// TIA Portal V18 export
FUNCTION "VerticalBeam_Main" : Void   // FC7, LAD
{ S7_Optimized_Access := 'TRUE' }
VERSION : 0.1
// stored: AutoNumber true, IsIECCheckEnabled false, SetENOAutomatically false, UDAEnableTagReadback false
BEGIN

REGION Network 1: 区域搜索
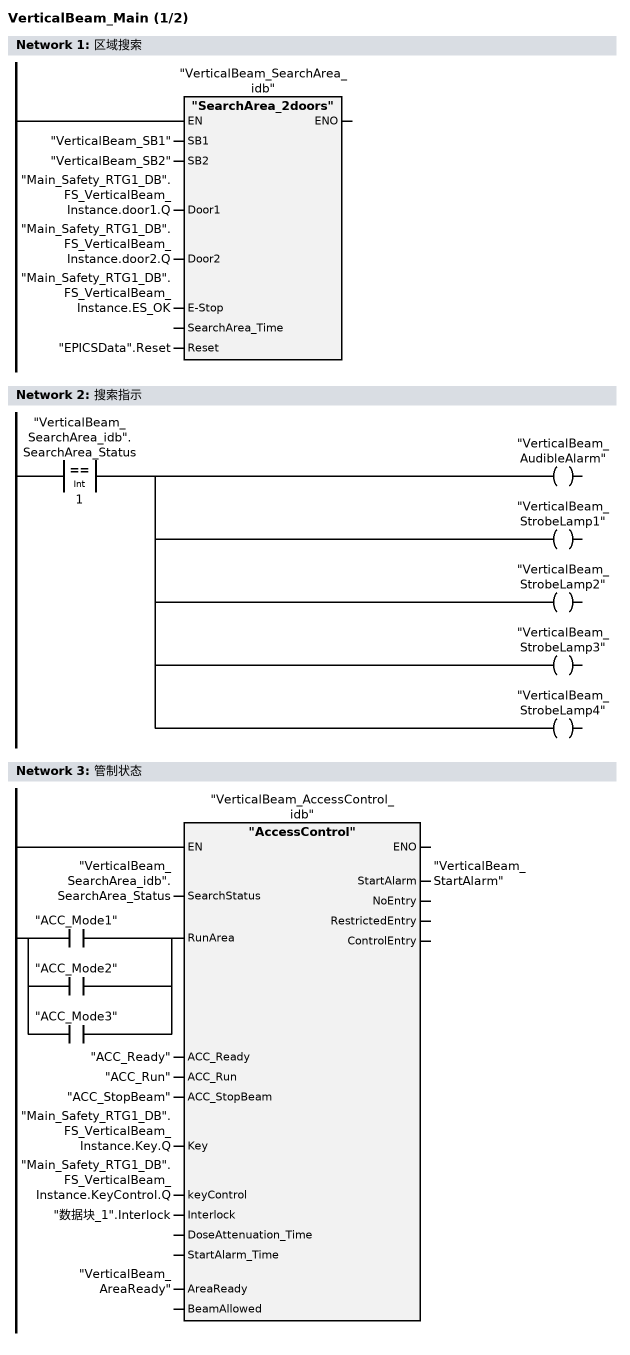
   RUNG wire#powerrail
      "VerticalBeam_SearchArea_idb"(SB1 := "VerticalBeam_SB1", SB2 := "VerticalBeam_SB2", Door1 := "Main_Safety_RTG1_DB".FS_VerticalBeam_Instance.door1.Q, Door2 := "Main_Safety_RTG1_DB".FS_VerticalBeam_Instance.door2.Q, "E-Stop" := "Main_Safety_RTG1_DB".FS_VerticalBeam_Instance.ES_OK, SearchArea_Time :=, Reset := "EPICSData".Reset)
   END_RUNG
   // the same network as SCL:
   "VerticalBeam_SearchArea_idb"(SB1 := "VerticalBeam_SB1",   // "SearchArea_2doors"
                           SB2 := "VerticalBeam_SB2",
                           Door1 := "Main_Safety_RTG1_DB".FS_VerticalBeam_Instance.door1.Q,
                           Door2 := "Main_Safety_RTG1_DB".FS_VerticalBeam_Instance.door2.Q,
                           "E-Stop" := "Main_Safety_RTG1_DB".FS_VerticalBeam_Instance.ES_OK,
                           Reset := "EPICSData".Reset);
END_REGION

REGION Network 2: 搜索指示
   RUNG wire#powerrail
      { S7_Templates := "SrcType := Int" } EQ_Contact(in1 := "VerticalBeam_SearchArea_idb".SearchArea_Status, in2 := 1)
      wire#w1
      Coil( "VerticalBeam_AudibleAlarm" )
   END_RUNG
   RUNG wire#w1
      Coil( "VerticalBeam_StrobeLamp1" )
   END_RUNG
   RUNG wire#w1
      Coil( "VerticalBeam_StrobeLamp2" )
   END_RUNG
   RUNG wire#w1
      Coil( "VerticalBeam_StrobeLamp3" )
   END_RUNG
   RUNG wire#w1
      Coil( "VerticalBeam_StrobeLamp4" )
   END_RUNG
   // the same network as SCL:
   "VerticalBeam_AudibleAlarm" := "VerticalBeam_SearchArea_idb".SearchArea_Status = 1;
   "VerticalBeam_StrobeLamp1" := "VerticalBeam_AudibleAlarm";
   "VerticalBeam_StrobeLamp2" := "VerticalBeam_AudibleAlarm";
   "VerticalBeam_StrobeLamp3" := "VerticalBeam_AudibleAlarm";
   "VerticalBeam_StrobeLamp4" := "VerticalBeam_AudibleAlarm";
END_REGION

REGION Network 3: 管制状态
   RUNG wire#powerrail
      "VerticalBeam_AccessControl_idb"(RunArea := wire#w1, SearchStatus := "VerticalBeam_SearchArea_idb".SearchArea_Status, ACC_Ready := "ACC_Ready", ACC_Run := "ACC_Run", ACC_StopBeam := "ACC_StopBeam", Key := "Main_Safety_RTG1_DB".FS_VerticalBeam_Instance.Key.Q, keyControl := "Main_Safety_RTG1_DB".FS_VerticalBeam_Instance.KeyControl.Q, Interlock := "数据块_1".Interlock, DoseAttenuation_Time :=, StartAlarm_Time :=, AreaReady := "VerticalBeam_AreaReady", BeamAllowed :=, StartAlarm => "VerticalBeam_StartAlarm", NoEntry =>, RestrictedEntry =>, ControlEntry =>)
   END_RUNG
   RUNG wire#powerrail
      Contact( "ACC_Mode1" )
   END_RUNG wire#w1
   RUNG wire#powerrail
      Contact( "ACC_Mode2" )
   END_RUNG wire#w1
   RUNG wire#powerrail
      Contact( "ACC_Mode3" )
   END_RUNG wire#w1
   // the same network as SCL:
   "VerticalBeam_AccessControl_idb"(SearchStatus := "VerticalBeam_SearchArea_idb".SearchArea_Status,   // "AccessControl"
                           RunArea := "ACC_Mode1" OR "ACC_Mode2" OR "ACC_Mode3",
                           ACC_Ready := "ACC_Ready",
                           ACC_Run := "ACC_Run",
                           ACC_StopBeam := "ACC_StopBeam",
                           Key := "Main_Safety_RTG1_DB".FS_VerticalBeam_Instance.Key.Q,
                           keyControl := "Main_Safety_RTG1_DB".FS_VerticalBeam_Instance.KeyControl.Q,
                           Interlock := "数据块_1".Interlock,
                           AreaReady := "VerticalBeam_AreaReady",
                           StartAlarm => "VerticalBeam_StartAlarm");
END_REGION

REGION Network 4: 管制输出
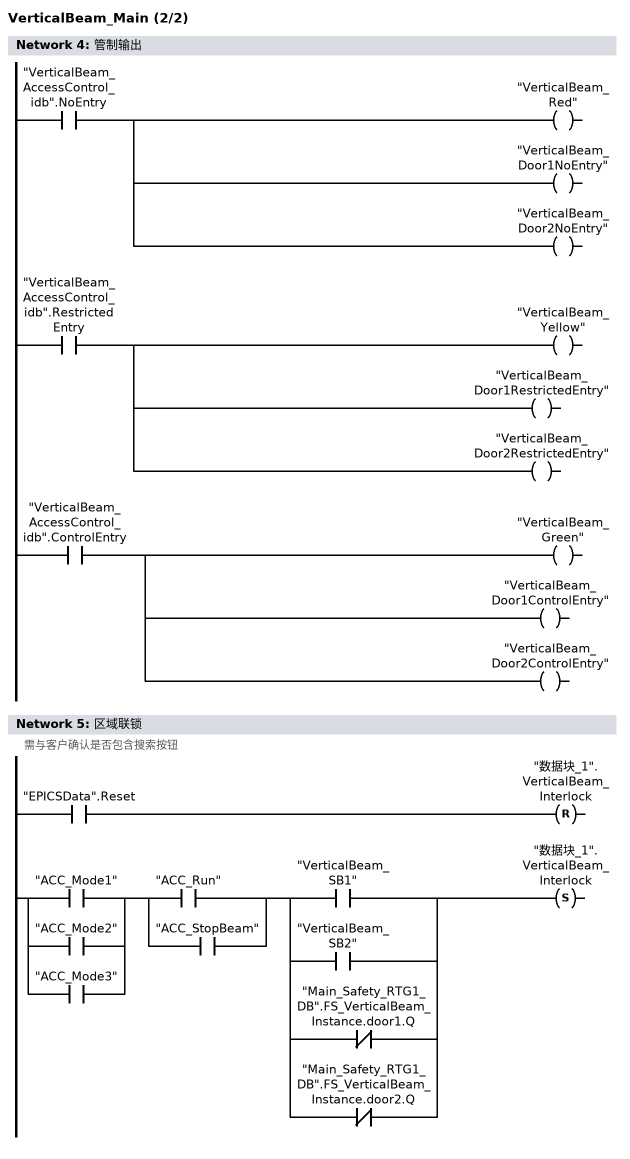
   RUNG wire#powerrail
      Contact( "VerticalBeam_AccessControl_idb".NoEntry )
      wire#w1
      Coil( "VerticalBeam_Red" )
   END_RUNG
   RUNG wire#w1
      Coil( "VerticalBeam_Door1NoEntry" )
   END_RUNG
   RUNG wire#w1
      Coil( "VerticalBeam_Door2NoEntry" )
   END_RUNG
   RUNG wire#powerrail
      Contact( "VerticalBeam_AccessControl_idb".RestrictedEntry )
      wire#w2
      Coil( "VerticalBeam_Yellow" )
   END_RUNG
   RUNG wire#w2
      Coil( "VerticalBeam_Door1RestrictedEntry" )
   END_RUNG
   RUNG wire#w2
      Coil( "VerticalBeam_Door2RestrictedEntry" )
   END_RUNG
   RUNG wire#powerrail
      Contact( "VerticalBeam_AccessControl_idb".ControlEntry )
      wire#w3
      Coil( "VerticalBeam_Green" )
   END_RUNG
   RUNG wire#w3
      Coil( "VerticalBeam_Door1ControlEntry" )
   END_RUNG
   RUNG wire#w3
      Coil( "VerticalBeam_Door2ControlEntry" )
   END_RUNG
   // the same network as SCL:
   "VerticalBeam_Red" := "VerticalBeam_AccessControl_idb".NoEntry;
   "VerticalBeam_Door1NoEntry" := "VerticalBeam_AccessControl_idb".NoEntry;
   "VerticalBeam_Door2NoEntry" := "VerticalBeam_AccessControl_idb".NoEntry;
   "VerticalBeam_Yellow" := "VerticalBeam_AccessControl_idb".RestrictedEntry;
   "VerticalBeam_Door1RestrictedEntry" := "VerticalBeam_AccessControl_idb".RestrictedEntry;
   "VerticalBeam_Door2RestrictedEntry" := "VerticalBeam_AccessControl_idb".RestrictedEntry;
   "VerticalBeam_Green" := "VerticalBeam_AccessControl_idb".ControlEntry;
   "VerticalBeam_Door1ControlEntry" := "VerticalBeam_AccessControl_idb".ControlEntry;
   "VerticalBeam_Door2ControlEntry" := "VerticalBeam_AccessControl_idb".ControlEntry;
END_REGION

REGION Network 5: 区域联锁
   // 需与客户确认是否包含搜索按钮
   RUNG wire#powerrail
      Contact( "EPICSData".Reset )
      R_Coil( "数据块_1".VerticalBeam_Interlock )
   END_RUNG
   RUNG wire#powerrail
      Contact( "ACC_Mode1" )
      wire#w1
      Contact( "ACC_Run" )
      wire#w2
      Contact( "VerticalBeam_SB1" )
      wire#w3
      S_Coil( "数据块_1".VerticalBeam_Interlock )
   END_RUNG
   RUNG wire#powerrail
      Contact( "ACC_Mode2" )
   END_RUNG wire#w1
   RUNG wire#powerrail
      Contact( "ACC_Mode3" )
   END_RUNG wire#w1
   RUNG wire#w1
      Contact( "ACC_StopBeam" )
   END_RUNG wire#w2
   RUNG wire#w2
      Contact( "VerticalBeam_SB2" )
   END_RUNG wire#w3
   RUNG wire#w2
      I_Contact( "Main_Safety_RTG1_DB".FS_VerticalBeam_Instance.door1.Q )
   END_RUNG wire#w3
   RUNG wire#w2
      I_Contact( "Main_Safety_RTG1_DB".FS_VerticalBeam_Instance.door2.Q )
   END_RUNG wire#w3
   // the same network as SCL:
   IF "EPICSData".Reset THEN "数据块_1".VerticalBeam_Interlock := FALSE; END_IF;
   IF ("ACC_Mode1" OR "ACC_Mode2" OR "ACC_Mode3") AND ("ACC_Run" OR "ACC_StopBeam") AND ("VerticalBeam_SB1" OR "VerticalBeam_SB2" OR NOT "Main_Safety_RTG1_DB".FS_VerticalBeam_Instance.door1.Q OR NOT "Main_Safety_RTG1_DB".FS_VerticalBeam_Instance.door2.Q) THEN
       "数据块_1".VerticalBeam_Interlock := TRUE;
   END_IF;
END_REGION
END_FUNCTION
